TEXTLIST TextList_Jog_mode
  0 = 'Slow'
  1 = 'Fast'
  2 = 'Continous'
  3 = 'Inching'
  4 = 'Inching Modulo'
   = ''
END_TEXTLIST

(* stored: Version 1.1.0.1, ProductVersion 3.1.4024.11
   TextList TextList_Jog_mode: Id {de32a786-6c96-49cb-8998-988727c6c539} *)
